// TIA Portal project "Recipe" (V13)

(* hardware
DEVICE "S7-1200 station_1"  S7-1200 Station
   slot 0: "Rack_0"  Rack  V1.0
   slot 1: "PLC_1"  CPU 1212C AC/DC/Rly  6ES7 212-1BE40-0XB0  V4.1
DEVICE "HMI_1"  KTP400 Basic PN
   slot 0: "HMI"  HMI  6AV2 123-2DB03-0AX0  13.0.1.0
   slot 1: "HMI_RT_1"  KTP400 Basic PN  6AV2 123-2DB03-0AX0  13.0.1.0
   slot 5: "HMI_1.IE_CP_1"  PROFINET Interface
      slot 1: "PROFINET Interface_1"  PROFINET Interface
         slot 1: "Port_1"  Port
*)

// ===== PLC "PLC_1"  CPU 1212C AC/DC/Rly =====

VAR_GLOBAL   // PLC tag table "Default tag table"
   "Tag_1" AT %MD5 : DWord;
   "Tag_2" AT %MD0 : DWord;
   "Tag_4" AT %MW5 : Word;
   "Tag_3" AT %MW10 : Int;
   "Tag_5" AT %M100.0 : Bool;
   "Warning light" AT %Q0.0 : Bool;
   "Tag_7" AT %M100.1 : Bool;
   "Tag_8" AT %Q0.1 : Bool;
   "Tag_9" AT %MD5 : Time;
   "Tag_10" AT %MD12 : Real;
   "Tag_11" AT %MW15 : Int;
   "Tag_12" AT %ID30 : DWord;
   "Tag_13" AT %MD22 : Real;
   "Tag_14" AT %MW50 : Word;
   "Tag_15" AT %Q0.2 : Bool;
   "Tag_16" AT %ID34 : DWord;
   "Tag_17" AT %MD25 : Real;
   "Tag_18" AT %MD26 : Real;
   "Fill Valve" AT %QD30 : Real;
   "Drain Valve" AT %QD34 : Real;
   "Tag_19" AT %M200.0 : Bool;
   "Tag_20" AT %M200.1 : Bool;
   "Animation bit" AT %M40.0 : Bool;
   "Clock_Byte" AT %MB300 : Byte;
   "Clock_10Hz" AT %M300.0 : Bool;
   "Clock_5Hz" AT %M300.1 : Bool;
   "Clock_2.5Hz" AT %M300.2 : Bool;
   "Clock_2Hz" AT %M300.3 : Bool;
   "Clock_1.25Hz" AT %M300.4 : Bool;
   "Clock_1Hz" AT %M300.5 : Bool;
   "Clock_0.625Hz" AT %M300.6 : Bool;
   "Clock_0.5Hz" AT %M300.7 : Bool;
   "Tag_21" AT %MB60 : Byte;
   "roller" AT %MD60 : Real;
   "roller_2" AT %MD70 : Real;
   "Tag_22" AT %MD65 : Real;
   "Tag_23" AT %MW60 : Int;
   "Tag_24" AT %MW65 : Int;
   "Down" AT %M90.0 : Bool;
   "Up" AT %M90.1 : Bool;
   "Tag_25" AT %MW75 : Int;
   "Tag_26" AT %MW78 : Int;
   "Tag_27" AT %MW80 : Int;
   "Alarm bit" AT %M99.0 : Bool;
   "Alarm register" AT %MW99 : Int;
   "OK bit" AT %M99.1 : Bool;
   "Reset Alarm" AT %M99.2 : Bool;
END_VAR

FUNCTION "MHJ-PLC-Lab-Function-S71200" : Void   // FC1, SCL
{ S7_Optimized_Access := 'FALSE' }
VERSION : 0.1
BEGIN

   #Value := PEEK(area := 16#82,
                  dbNumber := 0,
                  byteOffset := 511);
   #Value := #Value + 1;

   POKE(area := 16#82,
        dbNumber := 0,
        byteOffset := 511,
        value := #Value);

   POKE(area := 16#81,
        dbNumber := 0,
        byteOffset := 1016,
        value := #Value_01_DW);
   POKE(area := 16#81,
        dbNumber := 0,
        byteOffset := 1020,
        value := #Value_02_DW);

   POKE(area := 16#81,
        dbNumber := 0,
        byteOffset := 511,
        value := B#16#00);

   FOR #forVal := 0 TO 120 DO
       FOR #forVal_2 := 0 TO 10 DO
           #rdTimeReturn := RD_SYS_T(#outputTime);
           #rdTimeReturn := WR_SYS_T(#outputTime);
           #rdTimeReturn := RD_SYS_T(#outputTime);
           #rdTimeReturn := WR_SYS_T(#outputTime);
       END_FOR;
       #SyncVal := PEEK(area := 16#81,
                        dbNumber := 0,
                        byteOffset := 511);
       IF #SyncVal = #CompVal THEN
           GOTO M_1;
       END_IF;
   END_FOR;
   RETURN;

   M_1:
   POKE(area := 16#81,
        dbNumber := 0,
        byteOffset := 511,
        value := B#16#0);
END_FUNCTION

ORGANIZATION_BLOCK "Main"   // OB1, LAD, ProgramCycle
TITLE = "Main Program Sweep (Cycle)"
{ S7_Optimized_Access := 'FALSE' }
VERSION : 0.1
BEGIN

REGION Network 1
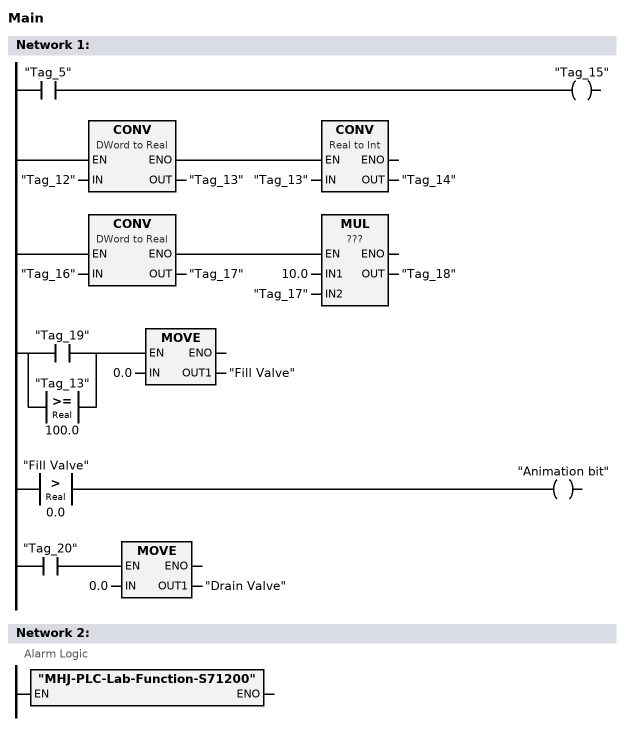
   RUNG wire#powerrail
      Contact( "Tag_5" )
      Coil( "Tag_15" )
   END_RUNG
   RUNG wire#powerrail
      { S7_Templates := "[SrcType := DWord, DestType := Real]"; S7_GenerateENO := "TRUE" } Convert(in := "Tag_12", out => "Tag_13")
      { S7_Templates := "[SrcType := Real, DestType := Int]"; S7_GenerateENO := "TRUE" } Convert(in := "Tag_13", out => "Tag_14")
   END_RUNG
   RUNG wire#powerrail
      { S7_Templates := "[SrcType := DWord, DestType := Real]"; S7_GenerateENO := "TRUE" } Convert(in := "Tag_16", out => "Tag_17")
      { S7_Templates := "SrcType := ???"; S7_GenerateENO := "TRUE" } Mul(in1 := 10.0, in2 := "Tag_17", out => "Tag_18")
   END_RUNG
   RUNG wire#powerrail
      Contact( "Tag_19" )
      wire#w1
      { S7_GenerateENO := "TRUE" } Move(in := 0.0, out1 => "Fill Valve")
   END_RUNG
   RUNG wire#powerrail
      { S7_Templates := "SrcType := Real" } GE_Contact(in1 := "Tag_13", in2 := 100.0)
   END_RUNG wire#w1
   RUNG wire#powerrail
      { S7_Templates := "SrcType := Real" } GT_Contact(in1 := "Fill Valve", in2 := 0.0)
      Coil( "Animation bit" )
   END_RUNG
   RUNG wire#powerrail
      Contact( "Tag_20" )
      { S7_GenerateENO := "TRUE" } Move(in := 0.0, out1 => "Drain Valve")
   END_RUNG
   // the same network as SCL:
   // ENO of a box is taken as its EN; it also drops when the box reports an error
   "Tag_15" := "Tag_5";
   "Tag_13" := DWORD_TO_REAL("Tag_12");
   "Tag_14" := REAL_TO_INT("Tag_13");
   "Tag_17" := DWORD_TO_REAL("Tag_16");
   "Tag_18" := 10.0 * "Tag_17";
   IF "Tag_19" OR ("Tag_13" >= 100.0) THEN "Fill Valve" := 0.0; END_IF;
   "Animation bit" := "Fill Valve" > 0.0;
   IF "Tag_20" THEN "Drain Valve" := 0.0; END_IF;
END_REGION

REGION Network 2
   // Alarm Logic
   RUNG wire#powerrail
      "MHJ-PLC-Lab-Function-S71200"()
   END_RUNG
   // the same network as SCL:
   "MHJ-PLC-Lab-Function-S71200"();
END_REGION
END_ORGANIZATION_BLOCK

(* ===== HMI "HMI_RT_1" =====
connection "HMI_Connection_1": ETHERNET, SMART_S7_1200_OMS

HMI tags "Default tag table"
   "Tag_5" : Bool = PLC "Tag_5", 100 ms
   "Tag_7" : Bool = PLC "Tag_7", 100 ms
   "Tag_6" : Bool = PLC "Warning light", 100 ms
   "Tag_10" : Real = PLC "Tag_10", 1 s
   "Tag_11" : Int = PLC "Tag_11", 1 s
   "Tag_14" : Word = PLC "Tag_14", 100 ms
   "Tag_17" : Real = PLC "Tag_17", 100 ms
   "Tag_18" : Real = PLC "Tag_18", 100 ms
   "Fill Valve" : Real = PLC "Fill Valve", 100 ms
   "Drain Valve" : Real = PLC "Drain Valve", 100 ms
   "Tag_19" : Bool = PLC "Tag_19", 100 ms
   "Tag_20" : Bool = PLC "Tag_20", 100 ms
   "Animation bit" : Bool = PLC "Animation bit", 1 s
   "Tag_13" : Real = PLC "Tag_13", 1 s
   "Tag_21" : Byte = PLC "Tag_21", 100 ms
   "roller_HMI" : Real = PLC "roller", 100 ms
   "roller_2" : Real = PLC "roller_2", 100 ms
   "Tag_23" : Int = PLC "Tag_23", 100 ms
   "Tag_25" : Int = PLC "Tag_25", 100 ms
   "Up" : Bool = PLC "Up", 100 ms
   "Alarm bit" : Bool = PLC "Alarm bit", 1 s
   "Alarm register" : Int = PLC "Alarm register", 1 s

discrete alarms
   1: '', class Warnings, trigger "Alarm register" bit 8
   2: '', class Warnings, trigger "Alarm register" bit 9

graphic list "Valve": 0 'OFF'; 1..7 'Partially ON_1'; 8..10 'ON_1'

graphic list "Pipes": 0 'not flowing'; 1..7 'Partially flowing'; 8..10 'flowing'

graphic list "Roller": 0..249 '1'; 250..499 '2'; 500..749 '3'; 750..1000 '4'

graphic list "Motor": 0 'Graphic_24'; 1 'Graphic_25'

graphic list "Arrow": 0 'Graphic_27'; 1 'Graphic_26'

Template "Template_1" 480x272
   Button "Template_Button" at 388,227 size 63x44
   Button "Template_Button_3" at 28,227 size 63x44

screen "Root screen" 480x272, template "Template_1"
   Button "Button_6" at 283,221 size 65x32
   TextField "Text field_1" at 148,76 size 273x32
   GraphicView "Graphic view_1" at 223,3 size 63x54
   TextField "Text field_2" at 100,57 size 336x27

screen "Tank" 480x272
   Bar "Bar_1" at 254,76 size 120x139
   TextField "Text field_2" at 248,1 size 135x23
   GraphicView "Graphic view_1" at 254,60 size 122x18
   GraphicView "Graphic view_2" at 253,213 size 123x28
   Button "Button_4" at 429,190 size 45x23
   IOField "I/O field_1" at 383,60 size 43x29
   IOField "I/O field_2" at 383,187 size 43x29
   Button "Button_3" at 429,63 size 45x23
   IOField "I/O field_3" at 378,133 size 43x18
   GraphicView "Graphic view_5" at 295,34 size 33x28
   GraphicIOField "Graphic I/O field_1" at 387,27 size 39x32
   GraphicIOField "Graphic I/O field_2" at 385,230 size 39x32
   GraphicIOField "Graphic I/O field_3" at 327,41 size 62x13
   GraphicIOField "Graphic I/O field_4" at 424,41 size 56x13
   GraphicIOField "Graphic I/O field_5" at 325,245 size 62x13
   GraphicIOField "Graphic I/O field_6" at 422,245 size 58x13
   TextField "Text field_3" at 422,132 size 23x22
   GraphicView "Graphic view_3" at 303,239 size 23x25
   Button "Button_1" at 12,227 size 67x32
   TrendView "Trend view_1" at 0,15 size 250x207
*)